FUNCTION_BLOCK inv
VAR_INPUT
	x: ARRAY[0..120] OF LREAL;
END_VAR
VAR_OUTPUT
	y: ARRAY[0..120] OF LREAL;
END_VAR
VAR
	i0_invNxN: invNxN;
END_VAR


i0_invNxN(x := x);
y := i0_invNxN.y;

END_FUNCTION_BLOCK

(* stored: Version 1.1.0.1, ProductVersion 3.1.4022.7
   POU inv: Id {43b477f3-cf64-427e-9d63-5a4c33a2c10e}, SpecialFunc None *)
